# B&R Automation Studio project laba001KRBO
Automation Studio 4.5.2.102

## Configuration laba001

### Task classes (Cpu.sw)
```
Cyclic#4:
  Main <- Main.prg
Libraries: Library
```

## Logical view

### Global.var - Global variables
```iecst
VAR
	integrator : FB_integrator;
	count : REAL;
	Enable : BOOL;
	speed : REAL;
	fb_motor : FB_motor;
	fb_motor2 : FB_motor;
	fb_controller : FB_regulator;
END_VAR
```

### Package Logical/Libraries - Global libraries

### Library Logical/Libraries/Library (ANSIC)

#### Library.fun - Exported functions and function blocks
```iecst
{REDUND_ERROR} FUNCTION_BLOCK FB_integrator (*TODO: Add your comment here*) (*$GROUP=User,$CAT=User,$GROUPICON=User.png,$CATICON=User.png*)
	VAR_INPUT
		in : REAL;
	END_VAR
	VAR_OUTPUT
		out : REAL;
	END_VAR
	VAR
		prev_state : REAL;
		dt : REAL;
	END_VAR
END_FUNCTION_BLOCK

{REDUND_ERROR} FUNCTION_BLOCK FB_motor (* *) (*$GROUP=User,$CAT=User,$GROUPICON=User.png,$CATICON=User.png*)
	VAR_INPUT
		u : REAL;
	END_VAR
	VAR_OUTPUT
		w : REAL;
		phi : REAL;
	END_VAR
	VAR
		integrator : FB_integrator;
		Tm : REAL;
		ke : REAL;
		dt : REAL;
	END_VAR
END_FUNCTION_BLOCK

{REDUND_ERROR} FUNCTION_BLOCK FB_regulator (*TODO: Add your comment here*) (*$GROUP=User,$CAT=User,$GROUPICON=User.png,$CATICON=User.png*)
	VAR_INPUT
		e : REAL;
	END_VAR
	VAR_OUTPUT
		u : REAL;
	END_VAR
	VAR
		k_p : REAL;
		k_i : REAL;
		integrator : FB_integrator;
		iyOld : REAL;
		max_abs_value : REAL;
		e_p : REAL;
		dt : REAL;
	END_VAR
END_FUNCTION_BLOCK
```

#### FB_integrator.c
```c
#include <bur/plctypes.h>
#ifdef __cplusplus
	extern "C"
	{
#endif
	#include "Library.h"
#ifdef __cplusplus
	};
#endif
/* TODO: Add your comment here */
void FB_integrator(struct FB_integrator* inst)
{
    inst->out+=inst->in;
}
```

#### FB_motor.c
```c
#include <bur/plctypes.h>
#ifdef __cplusplus
	extern "C"
	{
#endif
	#include "Library.h"
#ifdef __cplusplus
	};
#endif
void FB_motor(struct FB_motor* inst)
{
    inst->integrator.in = (inst->u*(1/inst->ke) - inst->w) * (inst->dt/inst->Tm);
    FB_integrator(&(inst->integrator));

    inst->w = inst->integrator.out;
    inst->integrator.in=inst->w*inst->dt;
    FB_integrator(&(inst->integrator));

    inst->phi=inst->integrator.out;
}
```

#### FB_regulator.c
```c
#include <bur/plctypes.h>
#ifdef __cplusplus
	extern "C"
	{
#endif
	#include "Library.h"
#ifdef __cplusplus
	};
#endif
/* TODO: Add your comment here */
void FB_regulator(struct FB_regulator* inst)
{
    inst->integrator.in=inst->e*inst->k_i*inst->dt+inst->iyOld;
    FB_integrator(&(inst->integrator));

    inst->e_p=inst->e*inst->k_p;

    if(inst->e_p < inst->max_abs_value || inst->e_p > -inst->max_abs_value);
    else{
        if (inst->e_p < 0) inst->e_p = inst->max_abs_value;
        else inst->e_p = -inst->max_abs_value;
    }
    inst->e_p += inst->integrator.out;
    if(inst->e_p < inst->max_abs_value || inst->e_p > -inst->max_abs_value)
        inst->u = inst->e_p;
    else{
        if(inst->e_p > 0) inst->u = inst->max_abs_value;
        else inst->u = -inst->max_abs_value;
    }
    inst->iyOld = inst->u - inst->e_p;
}
```

### Program Logical/Main (ANSIC)

#### Main.c
```c
#include <bur/plctypes.h>

#ifdef _DEFAULT_INCLUDES
#include <AsDefault.h>
#endif

void _INIT ProgramInit(void)
{
    Enable = 1;
    count = 0;
    speed = 0;

    fb_motor.dt = 0.005;
    fb_motor.ke = 2;
    fb_motor.Tm = 0.07;
    fb_motor2.dt = 0.005;
    fb_motor2.ke = 1;
    fb_motor2.Tm = 0.07;

    fb_controller.dt = 0.01;
    fb_controller.k_p = 1.4;
    fb_controller.k_i = 20;
    fb_controller.max_abs_value = 24;
}

void _CYCLIC ProgramCyclic(void)
{
    if(Enable == 1)
    {
        count += 10;
        if (count >= 500 && count <= 1000) speed = 40;
        else speed = 5;
    }
    else speed = 0;
    fb_controller.e = speed - fb_motor.w;
    fb_motor2.u = speed * fb_motor2.ke;
    fb_motor.u = fb_controller.u * fb_motor.ke;
    FB_motor(&fb_motor);
    FB_motor(&fb_motor2);
}

void _EXIT ProgramExit(void)
{

}
```

Listed in the project but not available here: Logical/Global.typ, Logical/Libraries/Library/Types.typ, Logical/Libraries/Library/Constants.var
